// TIA Portal V19 export
TYPE "UDT_VALVE"
   STRUCT
      cmd : Struct   // Control commands
         auto : Bool := false;   // Auto
         man : Bool := false;   // Manual
         main : Bool := false;   // Main route
         upper : Bool := false;   // Upper s/l route
         lower : Bool := false;   // Lower s/l route
         deact : Bool := false;   // Deactivated
      END_STRUCT;
      ind : Struct   // Control indications
         auto : Bool := false;   // Auto
         man : Bool := false;   // Manual
         main : Bool := false;   // Main route
         upper : Bool := false;   // Upper s/l route
         lower : Bool := false;   // Lower s/l route
         deact : Bool := false;   // Deactivated
      END_STRUCT;
      man : Struct   // Manual activations
         main : Bool := false;   // Main route
         upper : Bool := false;   // Upper s/l route
         lower : Bool := false;   // Lower s/l route
      END_STRUCT;
      sim : Struct   // Simulation
         main { S7_SetPoint := 'True'} : Bool := false;   // Activated main position
         upper { S7_SetPoint := 'True'} : Bool := false;   // Activated upper s/l position
         lower { S7_SetPoint := 'True'} : Bool := false;   // Activated lower s/l position
         deact { S7_SetPoint := 'True'} : Bool := false;   // Deactivated position
      END_STRUCT;
      faults : Struct   // Fault monitoring
         ftamain { S7_SetPoint := 'True'} : "UDT_ALARMACKN";   // Setpoint: failed to activate main route
         ftaupper { S7_SetPoint := 'True'} : "UDT_ALARMACKN";   // Setpoint: failed to activate upper s/l route
         ftalower { S7_SetPoint := 'True'} : "UDT_ALARMACKN";   // Setpoint: failed to activate lower s/l route
         ftd { S7_SetPoint := 'True'} : "UDT_ALARMACKN";   // Setpoint: failed to deactivate valve
         il { S7_SetPoint := 'True'} : "UDT_ALARMACKN";   // Setpoint: failed to deactivate valve
         fpreset : Bool := false;   // Faceplate reset for individual treatment
      END_STRUCT;
      delaymain { S7_SetPoint := 'True'} : "UDT_DELAYONOFF";   // Activation delay on/off for main route
      delayupper { S7_SetPoint := 'True'} : "UDT_DELAYONOFF";   // Activation delay on/off for upper s/l route
      delaylower { S7_SetPoint := 'True'} : "UDT_DELAYONOFF";   // Activation delay on/off for lower s/l route
      out : Struct   // Output
         actmain : Bool := false;   // Activate main route
         actupper : Bool := false;   // Activate upper s/l route
         actlower : Bool := false;   // Activate lower s/l route
      END_STRUCT;
      status : Struct   // Status
         vfbmain : Bool := false;   // Activated main route
         vfbupper : Bool := false;   // Activated upper s/l route
         vfblower : Bool := false;   // Activated lower s/l route
         vfbdeact : Bool := false;   // Deactivated
         fault : Bool := false;   // Collective fault
         ilactmain : Bool := false;   // Allow to activate main route
         ilactupper : Bool := false;   // Allow to activate upper s/l route
         ilactlower : Bool := false;   // Allow to activate lower s/l route
         icon : Int := 0;   // Valve's graphic icon
      END_STRUCT;
   END_STRUCT;
END_TYPE
